// TwinCAT 3 PLC project XMLServerTesten
// ProgramVersion: 3.1.4023.0
// libraries:
//   Tc2_Standard, * (Beckhoff Automation GmbH)
//   Tc2_System, * (Beckhoff Automation GmbH)
//   Tc2_Utilities, * (Beckhoff Automation GmbH)
//   Tc2_XmlDataSrv, * (Beckhoff Automation GmbH)
//   Tc3_Module, * (Beckhoff Automation GmbH)
// project tree:
//   DUTs/ Datensatz.TcDUT, ST_TimeDiff.TcDUT (not stored), XMLHeader.TcDUT (not stored)
//   / PlcTask.TcTTO (not stored)
//   POUs/ get_Diff.TcPOU (not stored), fileT_to_sysT.TcPOU, MAIN.TcPOU, RecordEndTime.TcPOU (not stored), RecordStartTime.TcPOU (not stored), write_to_Buffer.TcPOU (not stored), write_to_XML.TcPOU, DataLogging.TcPOU
// real-time tasks:
//   TASK PlcTask: cycle T#10ms, priority 20, ADS port 350

// ---- DUTs/Datensatz.TcDUT
TYPE Datensatz :
STRUCT
	Timestamp : STRING ;
	roomnum : REAL;
	temp : REAL;
	signal3 : REAL;
	signal4 : REAL;
	signal5 : REAL;
	signal6 : REAL;
	signal7 : REAL;
	signal8 : REAL;
END_STRUCT
END_TYPE

// ---- POUs/fileT_to_sysT.TcPOU
FUNCTION_BLOCK fileT_to_sysT
VAR_INPUT
	T_LoDW : DWORD;
	T_HiDW : DWORD;
END_VAR
VAR_OUTPUT
	sysT : TIMESTRUCT;
END_VAR
VAR
	fileT : T_FILETIME;
END_VAR

fileT.dwLowDateTime:= T_LoDW;			//change hex time to hh:mm:ss time
fileT.dwHighDateTime:= T_HiDW;
sysT := FILETIME_TO_SYSTEMTIME(fileT);

END_FUNCTION_BLOCK

// ---- POUs/MAIN.TcPOU
PROGRAM MAIN
VAR
	XMLTesten : DataLogging;
END_VAR

XMLTesten();

END_PROGRAM

// ---- POUs/DataLogging.TcPOU
FUNCTION_BLOCK DataLogging
VAR
	bBufferFinish : BOOL;
	bBufferFinish2 : BOOL;
	bXMLFinish : BOOL;
	RecordStartTime : RecordStartTime;
	write_to_Buffer : write_to_Buffer;
	RecordEndTime : RecordEndTime;
	write_to_XML : write_to_XML;
	write_to_XML2 : write_to_XML;
	get_Diff : get_Diff;
	XMLFileName : T_MaxString;
	XMLFileName2 : T_MaxString;
	Buffer1 : ARRAY[1..100] OF Datensatz;
	Buffer2 : ARRAY[1..100] OF Datensatz;
	Buffer : ARRAY[1..100] OF Datensatz;
	m: INT :=1;
	StopRecordStart: BOOL := TRUE;
	DownTrigDetect: F_TRIG;
	WriteTimeDiff: ST_TimeDiff;
	Name: T_MaxString;
	bExecute: BOOL := false;
	bXMLFinish2: BOOL;
	bExecute2: BOOL := false;
	l: STRING(255);
	TimestampSYS: TIMESTRUCT;
END_VAR

(*//record the start timestamp of writing to buffer
IF StopRecordStart THEN
	RecordStartTime(StartFlag := TRUE);
END_IF
StopRecordStart := FALSE; 			//be set so that the start timestamp is not refreshed when writing datensatz2

//when recordstarttime is finished the datensatz is written
IF RecordStartTime.RecordStFinish THEN*)

//start the function to get the needed to be recorded values
write_to_Buffer(TimestampSYS=>TimestampSYS,m := m,startrecord := TRUE);

//write first 100 values in Buffer1, second 100 values in buffer2
IF m < 100 THEN
	//RecordEndTime(EndFlag := TRUE);			//when 100 datensatz are written in buffer, record the end timestamp
	Buffer1[m]:= write_to_Buffer.Datensatz;
ELSIF m = 100 THEN
	bBufferFinish :=TRUE;
	Buffer1[m]:= write_to_Buffer.Datensatz;	
	l := CONCAT(CONCAT(WORD_TO_STRING(TimestampSYS.wYear),'-'),CONCAT(CONCAT(WORD_TO_STRING(TimestampSYS.wMonth),'-'),CONCAT(CONCAT(WORD_TO_STRING(TimestampSYS.wDay),'-'),CONCAT(CONCAT(WORD_TO_STRING(TimestampSYS.wHour),'-'),CONCAT(CONCAT(WORD_TO_STRING(TimestampSYS.wMinute),'-'),CONCAT(CONCAT(WORD_TO_STRING(TimestampSYS.wSecond),'-'),WORD_TO_STRING(TimestampSYS.wMilliseconds)))))));
ELSIF m < 200 THEN
	Buffer2[m-100]:= write_to_Buffer.Datensatz;	
ELSIF m = 200 THEN
	Buffer2[m-100]:= write_to_Buffer.Datensatz;
	bBufferFinish2 :=TRUE;
	m:=0;
	l := CONCAT(CONCAT(WORD_TO_STRING(TimestampSYS.wYear),'-'),CONCAT(CONCAT(WORD_TO_STRING(TimestampSYS.wMonth),'-'),CONCAT(CONCAT(WORD_TO_STRING(TimestampSYS.wDay),'-'),CONCAT(CONCAT(WORD_TO_STRING(TimestampSYS.wHour),'-'),CONCAT(CONCAT(WORD_TO_STRING(TimestampSYS.wMinute),'-'),CONCAT(CONCAT(WORD_TO_STRING(TimestampSYS.wSecond),'-'),WORD_TO_STRING(TimestampSYS.wMilliseconds)))))));
END_IF
m :=m+1;

	
//give name to xml files
Name:=CONCAT(CONCAT('C:\temp_Yizhen\',l),'TEST.xml');
XMLFileName := Name;
XMLFileName2 := Name;
//XMLFileName := 'C:\temp_Yizhen\Test.xml';


//write data from buffer to xml file
write_to_XML(WriteFinishFlag => bXMLFinish,sFilePath := XMLFileName,LogInput := Buffer1,bExecute := bExecute);
write_to_XML2(WriteFinishFlag => bXMLFinish2,sFilePath := XMLFileName2,LogInput := Buffer2,bExecute := bExecute2);

//reset write to xml function
IF bBufferFinish THEN
	bExecute := TRUE;
END_IF 

IF bBufferFinish2 THEN
	bExecute2 := TRUE;
END_IF 

IF bXMLFinish THEN
	bExecute := FALSE;
	bBufferFinish :=FALSE;
	bXMLFinish := FALSE;
END_IF

IF bXMLFinish2 THEN
	bExecute2 := FALSE;
	bBufferFinish2 :=FALSE;
	bXMLFinish2 := FALSE;
END_IF

(*//get timeintervall for writing into buffer (10ms*n)
get_Diff(WriteTimeDiff=>WriteTimeDiff,BeginLo := RecordStartTime.BeginLo,BeginHi := RecordStartTime.BeginHi,EndLo := RecordEndTime.EndLo, EndHi := RecordEndTime.EndHi);
*)

END_FUNCTION_BLOCK

// ---- POUs/write_to_XML.TcPOU
FUNCTION_BLOCK write_to_XML
VAR_INPUT
	LogInput : ARRAY[1..100] OF Datensatz;
	bExecute 		: BOOL := FALSE;
	sFilePath 	: T_MaxString := 'C:\temp_Yizhen\Test.xml';  			//disable for CE
  //sFilePath 	: T_MaxString := '\Hard Disk\Test.xml';		//enable for CE
END_VAR
VAR_OUTPUT
	WriteTimeDiff: ST_TimeDiff;
	WriteFinishFlag : BOOL;
END_VAR
VAR
	bBusy : BOOL;
	bExecuteValue 		: BOOL;
	get_Diff : get_Diff;
	XmlSrvWriteValue : FB_XmlSrvWrite;
    sXPathData 		: T_MaxString := '/datafromroom/datapart';
  	INPUT: int;
	Error: BOOL;
	ErrID: UDINT;
	MyTimer: getsystemtime;
	UpTrigDetect: R_TRIG;
	DownTrigDetect: F_TRIG;
	DownTrigDetectHeader: F_TRIG;
	fileT_to_sysT_Before: fileT_to_sysT;
	fileT_to_sysT_After: fileT_to_sysT;
	SysTimeBefore: TIMESTRUCT;
	SysTimeAfter: TIMESTRUCT;
	BeginLo: UDINT;
	BeginHi: UDINT;
	EndLo: UDINT;
	EndHi: UDINT;
	MyTimer2: getsystemtime;
	Header: XMLHeader;
	XmlSrvWriteHeader: FB_XmlSrvWrite;
	sXPathHeader: T_MaxString := '/datafromroom/Header';
END_VAR

(* 	Sample1 creates an XML-file under the path C:\Test.xml and writes value1 to it. 
	Existing file will be overwritten.
	FUNCTIONBLOCK: FB_XmlSrvWrite *)
(*	
//start to get system time	
MyTimer();

//detect the trigger: false to true
UpTrigDetect(CLK:=bExecute);*)

//reset buffer reading flag
WriteFinishFlag := FALSE;

//detect the trigger:true to false
DownTrigDetect(CLK:=XmlSrvWriteValue.bBusy);
DownTrigDetectHeader(CLK:=XmlSrvWriteHeader.bBusy);

(*
//record beginning Timestamp of writing period
IF UpTrigDetect.Q THEN
	BeginLo := MyTimer.timeLoDW;							
	BeginHi := MyTimer.timeHiDW;
END_IF
*)

//write the xml header
XmlSrvWriteHeader(
	nMode	:= XMLSRV_ADDMISSING, 
  pSymAddr	:= ADR(Header),
  cbSymSize	:= SIZEOF(Header), 
  sFilePath	:= sFilePath,
  sXPath	:= sXPathHeader,
  bExecute	:= bExecute
);

//when xml header is done, start to write the values
IF DownTrigDetectHeader.Q THEN
	bExecuteValue := TRUE;
END_IF

//write values to xml file	
XmlSrvWriteValue(
  nMode		:= XMLSRV_ADDMISSING, 
  pSymAddr	:= ADR(LogInput),
  cbSymSize	:= SIZEOF(LogInput), 
  sFilePath	:= sFilePath,
  sXPath	:= sXPathData,
  bExecute	:= bExecuteValue
);

Error := XmlSrvWriteValue.bError;
ErrID := XmlSrvWriteValue.nErrId;
bBusy := XmlSrvWriteValue.bBusy; 


//record ending Timestamp of writing period
IF DownTrigDetect.Q THEN
	WriteFinishFlag := TRUE;
	bExecute := FALSE;
	bExecuteValue := FALSE;
	//EndHi := MyTimer.timeHiDW;
	//EndLo := MyTimer.timeLoDW;							
END_IF

(*//get timeintervall for writing into xml file
get_Diff(BeginLo := BeginLo,BeginHi := BeginHi,EndLo := EndLo, EndHi := EndHi);
WriteTimeDiff:=get_Diff.WriteTimeDiff;*)

END_FUNCTION_BLOCK
